PROGRAM CountCurrentPosition
VAR
END_VAR

// ONLY COUNTING, NO SETTING MOTORS ON/OFF

// COUNT ROTATION:
IF IO.Initialized AND Automatic.MotorR.CurrentlyMoving AND IO.StepRotatonSwitch = 1 THEN
	IO.LEDGreen := 0;
	IF IO.MotorRotationDirection = 0 THEN
		Automatic.RotationPositionCurrent := Automatic.RotationPositionCurrent + 1;
		IF NOT IO.Switch THEN
			Automatic.RotationPositionAuto := Automatic.RotationPositionAuto + 1;
		END_IF
	ELSE
		Automatic.RotationPositionCurrent := Automatic.RotationPositionCurrent - 1;
		IF NOT IO.Switch THEN
			Automatic.RotationPositionAuto := Automatic.RotationPositionAuto - 1;
		END_IF
	END_IF
ELSE
	IO.LEDGreen := 1;
END_IF

// COUNT Extension:
IF IO.Initialized AND Automatic.MotorE.CurrentlyMoving AND IO.StepExtensionSwitch = 1 THEN
	IO.LEDGreen := 0;
	IF IO.MotorExtensionDirection = 0 THEN
		Automatic.ExtensionPositionCurrent := Automatic.ExtensionPositionCurrent + 1;
		IF NOT IO.Switch THEN
			Automatic.ExtensionPositionAuto := Automatic.ExtensionPositionAuto + 1;
		END_IF
	ELSE
		Automatic.ExtensionPositionCurrent := Automatic.ExtensionPositionCurrent - 1;
		IF NOT IO.Switch THEN
			Automatic.ExtensionPositionAuto := Automatic.ExtensionPositionAuto - 1;
		END_IF
	END_IF
ELSE
	IO.LEDGreen := 1;
END_IF

// COUNT Lifting:
IF IO.Initialized AND Automatic.MotorL.CurrentlyMoving AND IO.StepLiftingSwitch = 1 THEN
	IO.LEDGreen := 0;
	IF IO.MotorLiftingDirection = 0 THEN
		Automatic.LiftingPositionCurrent := Automatic.LiftingPositionCurrent + 1;
		IF NOT IO.Switch THEN
			Automatic.LiftingPositionAuto := Automatic.LiftingPositionAuto + 1;
		END_IF
	ELSE
		Automatic.LiftingPositionCurrent := Automatic.LiftingPositionCurrent - 1;
		IF NOT IO.Switch THEN
			Automatic.LiftingPositionAuto := Automatic.LiftingPositionAuto - 1;
		END_IF
	END_IF
ELSE
	IO.LEDGreen := 1;
END_IF

// COUNT Grip:
IF IO.Initialized AND Automatic.MotorG.CurrentlyMoving AND IO.StepGripSwitch = 1 THEN
	IO.LEDGreen := 0;
	IF IO.MotorGripDirection = 0 THEN
		Automatic.GripPositionCurrent := Automatic.GripPositionCurrent + 1;
		IF NOT IO.Switch THEN
			Automatic.GripPositionAuto := Automatic.GripPositionAuto + 1;
		END_IF
	ELSE
		Automatic.GripPositionCurrent := Automatic.GripPositionCurrent - 1;
		IF NOT IO.Switch THEN
			Automatic.GripPositionAuto := Automatic.GripPositionAuto - 1;
		END_IF
	END_IF
ELSE
	IO.LEDGreen := 1;
END_IF

END_PROGRAM

(* stored: Version 1.1.0.1, ProductVersion 3.1.4024.13
   POU CountCurrentPosition: Id {80975f91-8736-487a-b4c3-c190ec7e08bf}, SpecialFunc None *)
